Yaskawa INFORM job: PARK-POS-ZONE-4.JBI

/JOB
//NAME PARK-POS-ZONE-4
//POS
///NPOS 1,1,0,0,0,0
///TOOL 0
///POSTYPE PULSE
///PULSE
C00000=75016,-48988,-40123,-68352,57928,88844
BC00000=79980
//INST
///DATE 2018/11/01 11:07
///ATTR SC,RW
///GROUP1 RB1,BS1
///LVARS 1,0,0,0,0,0,0,0
NOP
*teach
DIN LB000 SOUT#(36)
IFTHEN LB000=0
	 SET B003 5
	 SETUALM 8000 "Robot is not in teach mode." 0
	 TIMER T=1.00
	 JUMP *teach
ENDIF
SET B003 0
MOVJ C00000 BC00000 VJ=5.00
END
